Staubli VAL3: realTimeComm.dtx

mdesc mNomSpeed
public sio sClient
